FUNCTION F_RESET_Event : BOOL
VAR_INPUT
	dwID									: DWORD;
	dtActTime								: DT;
END_VAR
VAR
	i										: DINT;
END_VAR

// Znajdz i wstaw date zakonczenia
FOR i := 1 TO GVL_EHS.diNoOfEvents DO
	IF 	GVL_EHSP.arrEvent[i].dwID = dwID THEN
		GVL_EHSP.arrEvent[i].dtDateEnd		:= dtActTime;
		EXIT;
	END_IF
END_FOR

END_FUNCTION

(* stored: Version 1.1.0.1, ProductVersion 3.1.4020.12
   POU F_RESET_Event: Id {1ad57179-0d76-4c36-bd42-d55d18672361}, SpecialFunc None *)
